{attribute addProperty BoxType "EJ2521-0224-0016"}
{attribute addProperty Id "ControlAT %Q*Control_A1EB0E501621Frequency_valueAT %Q*UINT16217"}
{attribute addProperty CRC "174198979"}
{attribute addProperty SizeInBites "32"}
{attribute addProperty SizeInBytes "4"}
TYPE PTO_Control_0A6210C3 :
STRUCT
	{attribute addProperty Name "Control"}
	Control AT %Q* : Control_A1EB0E50;
	{attribute addProperty Name "Frequency_value"}
	Frequency_value AT %Q* : UINT;
END_STRUCT
END_TYPE

(* stored: Version 1.2.0.0, ProductVersion 3.1.4024.9
   DUT PTO_Control_0A6210C3: Id {73e7101a-f122-40f5-9495-90649ab3cdc1} *)
